FUNCTION_BLOCK AdsTcpUnitEx
VAR_INPUT
	setMode : (SEND, QUEUE);
END_VAR
VAR_OUTPUT
	bBusy : BOOL;
	error : BOOL;
	errorID : UDINT;
END_VAR
VAR
	socketsArr : ARRAY[1..numSockets] OF POINTER TO AdsSocket; //use this to find a socket
	
	//declare all sockets here
	AREA_2 : AdsSocket := (PrgName := TO_STRING(AreaNum.AREA_2), AmsNetId := '', AmsPort := 851); //local socket, unused
	AREA_3 : AdsSocket := (PrgName := TO_STRING(AreaNum.AREA_3), AmsNetId := '3.0.131.216.1.1', AmsPort := 851); //placeholder NetId
END_VAR
VAR
	socket : REFERENCE TO AdsSocket;
	
	messageQueue : AdsMessageQueue;
	nextMessage : AdsMessage;
	
	mode : (SEND, QUEUE);
END_VAR
VAR CONSTANT
	numSockets : INT := 2;
END_VAR

(*
	this extended version of AdsTcp communication provides the option to dynamically generate ADS messages into a queue
		due to the significant stack memory requirements, the QUEUE model can only be used on systems with adjustable stack
		using QUEUE mode on panel PCs (CP66xx) or other mini controllers can freeze the system
		
	QUEUE mode:
		when a message is polled, a socket with the same recipient name is identified
			if the identified socket is ready to send, then the message is passed to the socket
			otherwise, the message is placed back into the queue
		if no socket with a matching name can be identified, then the message is discarded
		
	SEND mode:
		if a socket matching the recipient name is identified and it is not busy or in error state, then the message is passed
		
	sendMessage() specifies a recipient name and data contents, then checks the mode to determine how to handle the message
*)

fillSocketsArr();

IF messageQueue.isEmpty() THEN
	mode := setMode;
END_IF

blocks();

IF mode = QUEUE THEN
	pollAndSend();	
END_IF

METHOD PRIVATE blocks : BOOL
VAR_INPUT
END_VAR
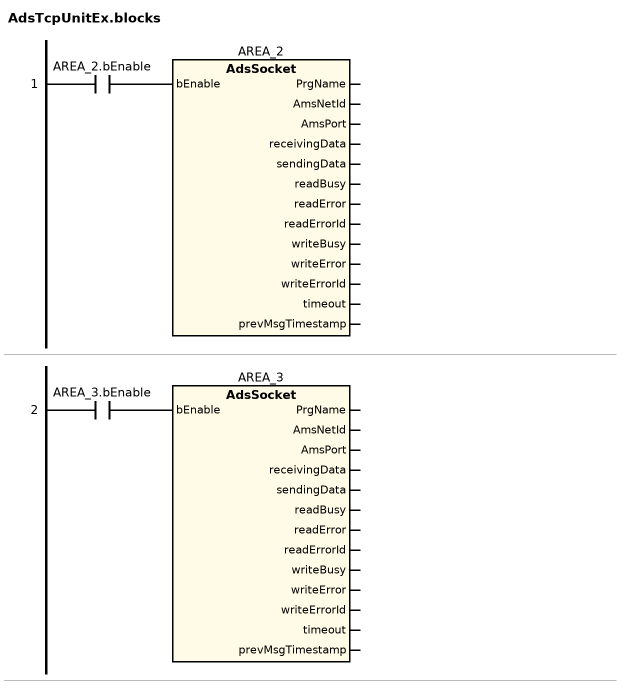
// NETWORK 1
AREA_2(bEnable := AREA_2.bEnable); // AdsSocket

// NETWORK 2
AREA_3(bEnable := AREA_3.bEnable); // AdsSocket
END_METHOD

METHOD fetchData : BOOL
VAR_INPUT
	senderName : STRING;
END_VAR
VAR_OUTPUT
	data : AdsData;
END_VAR
VAR
	i : INT;
END_VAR
FOR i:=1 TO numSockets BY 1 DO
	
	IF socketsArr[i]^.PrgName = senderName THEN
		fetchData := TRUE;
		data := socketsArr[i]^.receivingData;
		RETURN;
	END_IF
	
END_FOR
END_METHOD

METHOD PRIVATE fillSocketsArr : BOOL
VAR_INPUT
END_VAR
socketsArr[1] := ADR(AREA_2);
socketsArr[2] := ADR(AREA_3);
END_METHOD

METHOD PRIVATE findSocket : REFERENCE TO AdsSocket
VAR_INPUT
	recipient : STRING;
END_VAR
VAR
	i : INT;
END_VAR
FOR i:=1 TO numSockets BY 1 DO
	IF socketsArr[i] <> 0 AND_THEN socketsArr[i]^.PrgName = recipient THEN
		findSocket REF= socketsArr[i]^;
		RETURN;
	END_IF
END_FOR
END_METHOD

METHOD PRIVATE pollAndSend : BOOL
VAR_INPUT
END_VAR
nextMessage := messageQueue.poll(getSize => );
socket REF= findSocket(recipient := nextMessage.recipient);

IF __ISVALIDREF(socket) THEN
	
	IF NOT socket.writeBusy AND NOT socket.writeError AND socket.writeReady THEN
		socket.send(data := nextMessage.contents);
	ELSE //if socket is busy or has ERROR state, then message is returned to the end of the line
		messageQueue.push(value := nextMessage);
	END_IF
	
END_IF
END_METHOD

METHOD sendMessage : BOOL
VAR_INPUT
	recipient : STRING;
	data : REFERENCE TO AdsData;
END_VAR
VAR
	newMessage : AdsMessage;
END_VAR
CASE mode OF
	SEND:
		socket REF= findSocket(recipient := recipient);
		IF
			__ISVALIDREF(socket) AND_THEN
			NOT socket.writeBusy AND NOT socket.writeError
		THEN
			socket.send(data := data);
			sendMessage := TRUE;
		END_IF
	
	QUEUE:
		IF recipient <> '' THEN
			newMessage.recipient := recipient;
			newMessage.contents := data;
			
			sendMessage := messageQueue.push(newMessage);
		END_IF
	
END_CASE
END_METHOD

END_FUNCTION_BLOCK

(* stored: Version 1.1.0.1, ProductVersion 3.1.4024.11
   POU AdsTcpUnitEx: Id {fdbfe87f-1184-47dd-b08b-0750e1c8692f}, SpecialFunc None
   Folder Private: Id {81c0c8d6-6d0c-4d4e-a2d8-594730bd6eba}
   Method blocks: Id {fc203c2c-f273-4dce-94bc-433d9e033eb8}
   Method fetchData: Id {59b13f15-8c50-435f-aff0-1d930148d944}
   Method fillSocketsArr: Id {0e29de2e-63eb-4e68-a827-adcae2668ee8}
   Method findSocket: Id {d8b3993d-426a-4e5d-a36f-587468829b99}
   Method pollAndSend: Id {018dc648-0b60-4c81-a6e8-f9e64516fdaa}
   Method sendMessage: Id {20b0f168-c0bb-48be-90d8-084d1d464586} *)
